TYPE "KukaRobot_UserInput_1"
VERSION : 0.1
   STRUCT
      Public : Struct
         GI_TaskMode : USInt;
         GI_PartType : USInt;
         GI_SpeedSet : USInt;
         "GI_PosNo." : USInt;
         GI_5 : Byte;
         GI_6 : Byte;
         GI_7 : Byte;
         GI_8 : Byte;
         GI_9 : Byte;
         GI_10 : Byte;
      END_STRUCT;
      Gripper : Struct
         DI129_Grip1WP : Bool;
         DI130_Grip1HP : Bool;
         DI131_Grip2WP : Bool;
         DI132_Grip2HP : Bool;
         DI133_PartOnGrip1 : Bool;
         DI134_PartOnGrip2 : Bool;
         DI135 : Bool;
         DI136 : Bool;
         DI137 : Bool;
         DI138 : Bool;
         DI139 : Bool;
         DI140 : Bool;
         DI141 : Bool;
         DI142 : Bool;
         DI143 : Bool;
         DI144 : Bool;
         DI145 : Bool;
         DI146 : Bool;
         DI147 : Bool;
         DI148 : Bool;
         DI149 : Bool;
         DI150 : Bool;
         DI151 : Bool;
         DI152 : Bool;
         DI153 : Bool;
         DI154 : Bool;
         DI155 : Bool;
         DI156 : Bool;
         DI157 : Bool;
         DI158 : Bool;
         DI159 : Bool;
         DI160 : Bool;
      END_STRUCT;
      Home : Struct
         DI161_HomeSeqStart : Bool;
         DI162_AutoCycleStart : Bool;
         DI163 : Bool;
         DI164 : Bool;
         DI165 : Bool;
         DI166 : Bool;
         DI167 : Bool;
         DI168 : Bool;
         DI169_RobotMoved : Bool;
         DI170 : Bool;
         DI171 : Bool;
         DI172 : Bool;
         DI173 : Bool;
         DI174 : Bool;
         DI175 : Bool;
         DI176 : Bool;
         DI177_NG1_1 : Bool;
         DI178_NG1_2 : Bool;
         DI179_NG1_3 : Bool;
         DI180_NG1_4 : Bool;
         DI181_NG1_5 : Bool;
         DI182_NG2_1 : Bool;
         DI183_NG2_2 : Bool;
         DI184_NG2_3 : Bool;
         DI185_NG2_4 : Bool;
         DI186_NG2_5 : Bool;
         DI187_NG3_1 : Bool;
         DI188_NG3_2 : Bool;
         DI189_NG3_3 : Bool;
         DI190_NG3_4 : Bool;
         DI191_NG3_5 : Bool;
         DI192 : Bool;
      END_STRUCT;
      Special : Struct
         DI193 : Bool;
         DI194 : Bool;
         DI195 : Bool;
         DI196 : Bool;
         DI197 : Bool;
         DI198 : Bool;
         DI199 : Bool;
         DI200 : Bool;
         DI201 : Bool;
         DI202 : Bool;
         DI203 : Bool;
         DI204 : Bool;
         DI205 : Bool;
         DI206 : Bool;
         DI207 : Bool;
         DI208 : Bool;
         DI209 : Bool;
         DI210 : Bool;
         DI211 : Bool;
         DI212 : Bool;
         DI213 : Bool;
         DI214 : Bool;
         DI215 : Bool;
         DI216 : Bool;
         DI217 : Bool;
         DI218 : Bool;
         DI219 : Bool;
         DI220 : Bool;
         DI221 : Bool;
         DI222 : Bool;
         DI223 : Bool;
         DI224 : Bool;
      END_STRUCT;
      Cycle : Struct
         DI225_ScanPosReq : Bool;
         DI226_ScanPos1Complete : Bool;
         DI227_ScanPos2Complete : Bool;
         DI228_ScanPos3Complete : Bool;
         DI229_ScanPos4Complete : Bool;
         DI230_ScanPos5Complete : Bool;
         DI231_ScanPos6Complete : Bool;
         DI232_ScanPos7Complete : Bool;
         DI233 : Bool;
         DI234 : Bool;
         DI235 : Bool;
         DI236 : Bool;
         DI237 : Bool;
         DI238 : Bool;
         DI239 : Bool;
         DI240 : Bool;
         DI241_PickShaftPalletReq : Bool;   // 料盘Shaft取料请求
         DI242_ShaftNewPallet : Bool;   // 新料盘
         DI243 : Bool;
         DI244 : Bool;
         DI245 : Bool;
         DI246 : Bool;
         DI247 : Bool;
         DI248 : Bool;
         DI249_ShaftScanPutReq : Bool;   // Shaft读码放料请求  4#区域
         "DI250_" : Bool;
         "DI251_" : Bool;
         "DI252_" : Bool;
         DI253_ShaftScanPickReq : Bool;   // Shaft读码取料请求  4#区域
         "DI254_" : Bool;
         "DI255_" : Bool;
         "DI256_" : Bool;
         DI257_TableRingPickReq : Bool;   // 转台Ring取料请求  2#区域
         "DI258_" : Bool;
         "DI259_" : Bool;
         "DI260_" : Bool;
         DI261_RingScanReq : Bool;   // Ring扫码请求
         DI262_RingScanComplete : Bool;   // Ring扫码完成
         "DI263_" : Bool;
         "DI264_" : Bool;
         DI265_LoadPressNGReq1 : Bool;   // NG放料请求1 压装NG
         DI266_LoadShaftScanNGReq2 : Bool;   // NG放料请求2 Shaft读码NG
         DI267_LoadRingScanNGReq3 : Bool;   // NG放料请求3 Ring读码NG
         "DI268_" : Bool;
         "DI269_" : Bool;
         "DI270_" : Bool;
         "DI271_" : Bool;
         "DI272_" : Bool;
         DI273_PressShaftPutReq : Bool;   // Shaft压机放料请求  压机下方
         "DI274_" : Bool;
         "DI275_" : Bool;
         "DI276_" : Bool;
         DI277_PressRingPutReq : Bool;   // Ring压机放料请求   压机上面
         DI278_PressRingPutLeave : Bool;   // 压机2固定好产品，机器人可以离开
         "DI279_" : Bool;
         "DI280_" : Bool;
         DI281_PressPickShaftReq : Bool;   // 压机取料
         "DI282_" : Bool;
         "DI283_" : Bool;
         "DI284_" : Bool;
         "DI285_" : Bool;
         "DI286_" : Bool;
         "DI287_" : Bool;
         "DI288_" : Bool;
         DI289_GluePutReq : Bool;   // 点胶放料请求
         DI290 : Bool;
         DI291 : Bool;
         DI292 : Bool;
         DI293 : Bool;
         DI294 : Bool;
         DI295 : Bool;
         DI296 : Bool;
         DI297_MaintainRequest : Bool;
         DI298 : Bool;
         DI299 : Bool;
         DI300_HomeRequest : Bool;
         DI301 : Bool;
         DI302 : Bool;
         DI303 : Bool;
         DI304 : Bool;
         DI305_GripScan : Bool;
         DI306_ScanPartComplete : Bool;
         DI307_ScanPartFinish : Bool;
         DI308 : Bool;
         DI309 : Bool;
         DI310 : Bool;
         DI311 : Bool;
         DI312 : Bool;
         DI313 : Bool;
         DI314 : Bool;
         DI315 : Bool;
         DI316 : Bool;
         DI317 : Bool;
         DI318 : Bool;
         DI319 : Bool;
         DI320 : Bool;
         DI321 : Bool;
         DI322 : Bool;
         DI323 : Bool;
         DI324 : Bool;
         DI325 : Bool;
         DI326 : Bool;
         DI327 : Bool;
         DI328 : Bool;
         DI329 : Bool;
         DI330 : Bool;
         DI331 : Bool;
         DI332 : Bool;
         DI333 : Bool;
         DI334 : Bool;
         DI335 : Bool;
         DI336 : Bool;
         Camera_Y : DInt;
         Camera_Z : DInt;
         Camera_R : DInt;
      END_STRUCT;
      Safety : Struct
         DI433 : Bool;
         DI434 : Bool;
         DI435 : Bool;
         DI436 : Bool;
         DI437 : Bool;
         DI438 : Bool;
         DI439 : Bool;
         DI440 : Bool;
         DI441 : Bool;
         DI442 : Bool;
         DI443 : Bool;
         DI444 : Bool;
         DI445 : Bool;
         DI446 : Bool;
         DI447 : Bool;
         DI448 : Bool;
         DI449 : Bool;
         DI450 : Bool;
         DI451 : Bool;
         DI452 : Bool;
         DI453 : Bool;
         DI454 : Bool;
         DI455 : Bool;
         DI456 : Bool;
         DI457 : Bool;
         DI458 : Bool;
         DI459 : Bool;
         DI460 : Bool;
         DI461 : Bool;
         DI462 : Bool;
         DI463 : Bool;
         DI464 : Bool;
         DI465 : Bool;
         DI466 : Bool;
         DI467 : Bool;
         DI468 : Bool;
         DI469 : Bool;
         DI470 : Bool;
         DI471 : Bool;
         DI472 : Bool;
         DI473 : Bool;
         DI474 : Bool;
         DI475 : Bool;
         DI476 : Bool;
         DI477 : Bool;
         DI478 : Bool;
         DI479 : Bool;
         DI480 : Bool;
         DI481 : Bool;
         DI482 : Bool;
         DI483 : Bool;
         DI484 : Bool;
         DI485 : Bool;
         DI486 : Bool;
         DI487 : Bool;
         DI488 : Bool;
         DI489 : Bool;
         DI490 : Bool;
         DI491 : Bool;
         DI492 : Bool;
         DI493 : Bool;
         DI494 : Bool;
         DI495 : Bool;
         DI496 : Bool;
         DI497 : Bool;
         DI498 : Bool;
         DI499 : Bool;
         DI500 : Bool;
         DI501 : Bool;
         DI502 : Bool;
         DI503 : Bool;
         DI504 : Bool;
         DI505 : Bool;
         DI506 : Bool;
         DI507 : Bool;
         DI508 : Bool;
         DI509 : Bool;
         DI510 : Bool;
         DI511 : Bool;
         DI512 : Bool;
      END_STRUCT;
   END_STRUCT;

END_TYPE

